 X = -102.6 mm, Y = 123.5 mm, Z = 131.1 mm,       W = 0.0 deg, P = 0.0 deg,
    GP2:
        UF : 1, UT : 2,
       J1 = 0.0 deg, J2 = 0.0 deg
 };
P[160] {
    GP1:
        UF : 6, UT : 5,     CONFIG: 'N U T, 0, 0, 0',
       X = -119.0 mm, Y = 51.8 mm, Z = 131.1 mm,
       W = 0.0 deg, P = 0.0 deg,
    GP2:
        UF : 1, UT : 2,
       J1 = 0.0 deg, J2 = 0.0 deg
 };
P[356] {
    GP1:
        UF : 6, UT : 5,     CONFIG: 'N U T, 0, 0, 0',
 X = -102.0 mm, Y = 122.8 mm, Z = 131.1 mm,       W = 0.0 deg, P = 0.0 deg,
    GP2:
        UF : 1, UT : 2,
       J1 = 0.0 deg, J2 = 0.0 deg
 };
P[161] {
    GP1:
        UF : 6, UT : 5,     CONFIG: 'N U T, 0, 0, 0',
       X = -118.5 mm, Y = 51.0 mm, Z = 131.1 mm,
       W = 0.0 deg, P = 0.0 deg,
    GP2:
        UF : 1, UT : 2,
       J1 = 0.0 deg, J2 = 0.0 deg
 };
P[357] {
    GP1:
        UF : 6, UT : 5,     CONFIG: 'N U T, 0, 0, 0',
 X = -101.5 mm, Y = 122.0 mm, Z = 131.1 mm,       W = 0.0 deg, P = 0.0 deg,
    GP2:
        UF : 1, UT : 2,
       J1 = 0.0 deg, J2 = 0.0 deg
 };
P[162] {
    GP1:
        UF : 6, UT : 5,     CONFIG: 'N U T, 0, 0, 0',
       X = -117.9 mm, Y = 49.9 mm, Z = 131.1 mm,
       W = 0.0 deg, P = 0.0 deg,
    GP2:
        UF : 1, UT : 2,
       J1 = 0.0 deg, J2 = 0.0 deg
 };
P[358] {
    GP1:
        UF : 6, UT : 5,     CONFIG: 'N U T, 0, 0, 0',
 X = -100.9 mm, Y = 120.9 mm, Z = 131.1 mm,       W = 0.0 deg, P = 0.0 deg,
    GP2:
        UF : 1, UT : 2,
       J1 = 0.0 deg, J2 = 0.0 deg
 };
P[163] {
    GP1:
        UF : 6, UT : 5,     CONFIG: 'N U T, 0, 0, 0',
       X = -117.5 mm, Y = 48.5 mm, Z = 131.1 mm,
       W = 0.0 deg, P = 0.0 deg,
    GP2:
        UF : 1, UT : 2,
       J1 = 0.0 deg, J2 = 0.0 deg
 };
P[359] {
    GP1:
        UF : 6, UT : 5,     CONFIG: 'N U T, 0, 0, 0',
 X = -100.5 mm, Y = 119.5 mm, Z = 131.1 mm,       W = 0.0 deg, P = 0.0 deg,
    GP2:
        UF : 1, UT : 2,
       J1 = 0.0 deg, J2 = 0.0 deg
 };
P[164] {
    GP1:
        UF : 6, UT : 5,     CONFIG: 'N U T, 0, 0, 0',
       X = -116.9 mm, Y = 46.0 mm, Z = 131.1 mm,
       W = 0.0 deg, P = 0.0 deg,
    GP2:
        UF : 1, UT : 2,
       J1 = 0.0 deg, J2 = 0.0 deg
 };
P[360] {
    GP1:
        UF : 6, UT : 5,     CONFIG: 'N U T, 0, 0, 0',
 X = -99.9 mm, Y = 117.0 mm, Z = 131.1 mm,       W = 0.0 deg, P = 0.0 deg,
    GP2:
        UF : 1, UT : 2,
       J1 = 0.0 deg, J2 = 0.0 deg
 };
P[165] {
    GP1:
        UF : 6, UT : 5,     CONFIG: 'N U T, 0, 0, 0',
       X = -116.5 mm, Y = 42.8 mm, Z = 131.1 mm,
       W = 0.0 deg, P = 0.0 deg,
    GP2:
        UF : 1, UT : 2,
       J1 = 0.0 deg, J2 = 0.0 deg
 };
P[361] {
    GP1:
        UF : 6, UT : 5,     CONFIG: 'N U T, 0, 0, 0',
 X = -99.5 mm, Y = 113.8 mm, Z = 131.1 mm,       W = 0.0 deg, P = 0.0 deg,
    GP2:
        UF : 1, UT : 2,
       J1 = 0.0 deg, J2 = 0.0 deg
 };
P[166] {
    GP1:
        UF : 6, UT : 5,     CONFIG: 'N U T, 0, 0, 0',
       X = -115.8 mm, Y = 37.9 mm, Z = 131.1 mm,
       W = 0.0 deg, P = 0.0 deg,
    GP2:
        UF : 1, UT : 2,
       J1 = 0.0 deg, J2 = 0.0 deg
 };
P[362] {
    GP1:
        UF : 6, UT : 5,     CONFIG: 'N U T, 0, 0, 0',
 X = -98.8 mm, Y = 108.9 mm, Z = 131.1 mm,       W = 0.0 deg, P = 0.0 deg,
    GP2:
        UF : 1, UT : 2,
       J1 = 0.0 deg, J2 = 0.0 deg
 };
P[167] {
    GP1:
        UF : 6, UT : 5,     CONFIG: 'N U T, 0, 0, 0',
       X = -114.5 mm, Y = 27.9 mm, Z = 131.1 mm,
       W = 0.0 deg, P = 0.0 deg,
    GP2:
        UF : 1, UT : 2,
       J1 = 0.0 deg, J2 = 0.0 deg
 };
P[363] {
    GP1:
        UF : 6, UT : 5,     CONFIG: 'N U T, 0, 0, 0',
 X = -97.5 mm, Y = 98.9 mm, Z = 131.1 mm,       W = 0.0 deg, P = 0.0 deg,
    GP2:
        UF : 1, UT : 2,
       J1 = 0.0 deg, J2 = 0.0 deg
 };
P[168] {
    GP1:
        UF : 6, UT : 5,     CONFIG: 'N U T, 0, 0, 0',
       X = -113.4 mm, Y = 18.0 mm, Z = 131.1 mm,
       W = 0.0 deg, P = 0.0 deg,
    GP2:
        UF : 1, UT : 2,
       J1 = 0.0 deg, J2 = 0.0 deg
 };
P[364] {
    GP1:
        UF : 6, UT : 5,     CONFIG: 'N U T, 0, 0, 0',
 X = -96.4 mm, Y = 89.0 mm, Z = 131.1 mm,       W = 0.0 deg, P = 0.0 deg,
    GP2:
        UF : 1, UT : 2,
       J1 = 0.0 deg, J2 = 0.0 deg
 };
P[169] {
    GP1:
        UF : 6, UT : 5,     CONFIG: 'N U T, 0, 0, 0',
       X = -112.4 mm, Y = 8.1 mm, Z = 131.1 mm,
       W = 0.0 deg, P = 0.0 deg,
    GP2:
        UF : 1, UT : 2,
       J1 = 0.0 deg, J2 = 0.0 deg
 };
P[365] {
    GP1:
        UF : 6, UT : 5,     CONFIG: 'N U T, 0, 0, 0',
 X = -95.4 mm, Y = 79.1 mm, Z = 131.1 mm,       W = 0.0 deg, P = 0.0 deg,
    GP2:
        UF : 1, UT : 2,
       J1 = 0.0 deg, J2 = 0.0 deg
 };
P[170] {
    GP1:
        UF : 6, UT : 5,     CONFIG: 'N U T, 0, 0, 0',
       X = -111.6 mm, Y = -1.9 mm, Z = 131.1 mm,
       W = 0.0 deg, P = 0.0 deg,
    GP2:
        UF : 1, UT : 2,
       J1 = 0.0 deg, J2 = 0.0 deg
 };
P[366] {
    GP1:
        UF : 6, UT : 5,     CONFIG: 'N U T, 0, 0, 0',
 X = -94.6 mm, Y = 69.1 mm, Z = 131.1 mm,       W = 0.0 deg, P = 0.0 deg,
    GP2:
        UF : 1, UT : 2,
       J1 = 0.0 deg, J2 = 0.0 deg
 };
P[171] {
    GP1:
        UF : 6, UT : 5,     CONFIG: 'N U T, 0, 0, 0',
       X = -110.9 mm, Y = -11.9 mm, Z = 131.1 mm,
       W = 0.0 deg, P = 0.0 deg,
    GP2:
        UF : 1, UT : 2,
       J1 = 0.0 deg, J2 = 0.0 deg
 };
P[367] {
    GP1:
        UF : 6, UT : 5,     CONFIG: 'N U T, 0, 0, 0',
 X = -93.9 mm, Y = 59.1 mm, Z = 131.1 mm,       W = 0.0 deg, P = 0.0 deg,
    GP2:
        UF : 1, UT : 2,
       J1 = 0.0 deg, J2 = 0.0 deg
 };
P[172] {
    GP1:
        UF : 6, UT : 5,     CONFIG: 'N U T, 0, 0, 0',
       X = -110.3 mm, Y = -21.9 mm, Z = 131.1 mm,
       W = 0.0 deg, P = 0.0 deg,
    GP2:
        UF : 1, UT : 2,
       J1 = 0.0 deg, J2 = 0.0 deg
 };
P[368] {
    GP1:
        UF : 6, UT : 5,     CONFIG: 'N U T, 0, 0, 0',
 X = -93.3 mm, Y = 49.1 mm, Z = 131.1 mm,       W = 0.0 deg, P = 0.0 deg,
    GP2:
        UF : 1, UT : 2,
       J1 = 0.0 deg, J2 = 0.0 deg
 };
P[173] {
    GP1:
        UF : 6, UT : 5,     CONFIG: 'N U T, 0, 0, 0',
       X = -110.1 mm, Y = -24.0 mm, Z = 131.1 mm,
       W = 0.0 deg, P = 0.0 deg,
    GP2:
        UF : 1, UT : 2,
       J1 = 0.0 deg, J2 = 0.0 deg
 };
P[369] {
    GP1:
        UF : 6, UT : 5,     CONFIG: 'N U T, 0, 0, 0',
 X = -93.1 mm, Y = 47.0 mm, Z = 131.1 mm,       W = 0.0 deg, P = 0.0 deg,
    GP2:
        UF : 1, UT : 2,
       J1 = 0.0 deg, J2 = 0.0 deg
 };
P[174] {
    GP1:
        UF : 6, UT : 5,     CONFIG: 'N U T, 0, 0, 0',
       X = -109.5 mm, Y = -26.0 mm, Z = 131.1 mm,
       W = 0.0 deg, P = 0.0 deg,
    GP2:
        UF : 1, UT : 2,
       J1 = 0.0 deg, J2 = 0.0 deg
 };
P[370] {
    GP1:
        UF : 6, UT : 5,     CONFIG: 'N U T, 0, 0, 0',
 X = -92.5 mm, Y = 45.0 mm, Z = 131.1 mm,       W = 0.0 deg, P = 0.0 deg,
    GP2:
        UF : 1, UT : 2,
       J1 = 0.0 deg, J2 = 0.0 deg
 };
P[175] {
    GP1:
        UF : 6, UT : 5,     CONFIG: 'N U T, 0, 0, 0',
       X = -108.7 mm, Y = -28.0 mm, Z = 131.1 mm,
       W = 0.0 deg, P = 0.0 deg,
    GP2:
        UF : 1, UT : 2,
       J1 = 0.0 deg, J2 = 0.0 deg
 };
P[371] {
    GP1:
        UF : 6, UT : 5,     CONFIG: 'N U T, 0, 0, 0',
 X = -91.7 mm, Y = 43.0 mm, Z = 131.1 mm,       W = 0.0 deg, P = 0.0 deg,
    GP2:
        UF : 1, UT : 2,
       J1 = 0.0 deg, J2 = 0.0 deg
 };
P[176] {
    GP1:
        UF : 6, UT : 5,     CONFIG: 'N U T, 0, 0, 0',
       X = -107.0 mm, Y = -30.9 mm, Z = 131.1 mm,
       W = 0.0 deg, P = 0.0 deg,
    GP2:
        UF : 1, UT : 2,
       J1 = 0.0 deg, J2 = 0.0 deg
 };
P[372] {
    GP1:
        UF : 6, UT : 5,     CONFIG: 'N U T, 0, 0, 0',
 X = -90.0 mm, Y = 40.1 mm, Z = 131.1 mm,       W = 0.0 deg, P = 0.0 deg,
    GP2:
        UF : 1, UT : 2,
       J1 = 0.0 deg, J2 = 0.0 deg
 };
P[177] {
    GP1:
        UF : 6, UT : 5,     CONFIG: 'N U T, 0, 0, 0',
       X = -103.8 mm, Y = -36.3 mm, Z = 131.1 mm,
       W = 0.0 deg, P = 0.0 deg,
    GP2:
        UF : 1, UT : 2,
       J1 = 0.0 deg, J2 = 0.0 deg
 };
P[373] {
    GP1:
        UF : 6, UT : 5,     CONFIG: 'N U T, 0, 0, 0',
 X = -86.8 mm, Y = 34.7 mm, Z = 131.1 mm,       W = 0.0 deg, P = 0.0 deg,
    GP2:
        UF : 1, UT : 2,
       J1 = 0.0 deg, J2 = 0.0 deg
 };
P[178] {
    GP1:
        UF : 6, UT : 5,     CONFIG: 'N U T, 0, 0, 0',
       X = -102.7 mm, Y = -38.0 mm, Z = 131.1 mm,
       W = 0.0 deg, P = 0.0 deg,
    GP2:
        UF : 1, UT : 2,
       J1 = 0.0 deg, J2 = 0.0 deg
 };
P[374] {
    GP1:
        UF : 6, UT : 5,     CONFIG: 'N U T, 0, 0, 0',
 X = -85.7 mm, Y = 33.0 mm, Z = 131.1 mm,       W = 0.0 deg, P = 0.0 deg,
    GP2:
        UF : 1, UT : 2,
       J1 = 0.0 deg, J2 = 0.0 deg
 };
P[179] {
    GP1:
        UF : 6, UT : 5,     CONFIG: 'N U T, 0, 0, 0',
       X = -101.2 mm, Y = -39.4 mm, Z = 131.1 mm,
       W = 0.0 deg, P = 0.0 deg,
    GP2:
        UF : 1, UT : 2,
       J1 = 0.0 deg, J2 = 0.0 deg
 };
P[375] {
    GP1:
        UF : 6, UT : 5,     CONFIG: 'N U T, 0, 0, 0',
 X = -84.2 mm, Y = 31.6 mm, Z = 131.1 mm,       W = 0.0 deg, P = 0.0 deg,
    GP2:
        UF : 1, UT : 2,
       J1 = 0.0 deg, J2 = 0.0 deg
 };
P[180] {
    GP1:
        UF : 6, UT : 5,     CONFIG: 'N U T, 0, 0, 0',
       X = -99.8 mm, Y = -40.1 mm, Z = 131.1 mm,
       W = 0.0 deg, P = 0.0 deg,
    GP2:
        UF : 1, UT : 2,
       J1 = 0.0 deg, J2 = 0.0 deg
 };
P[376] {
    GP1:
        UF : 6, UT : 5,     CONFIG: 'N U T, 0, 0, 0',
 X = -82.8 mm, Y = 30.9 mm, Z = 131.1 mm,       W = 0.0 deg, P = 0.0 deg,
    GP2:
        UF : 1, UT : 2,
       J1 = 0.0 deg, J2 = 0.0 deg
 };
P[181] {
    GP1:
        UF : 6, UT : 5,     CONFIG: 'N U T, 0, 0, 0',
       X = -98.3 mm, Y = -40.7 mm, Z = 131.1 mm,
       W = 0.0 deg, P = 0.0 deg,
    GP2:
        UF : 1, UT : 2,
       J1 = 0.0 deg, J2 = 0.0 deg
 };
P[377] {
    GP1:
        UF : 6, UT : 5,     CONFIG: 'N U T, 0, 0, 0',
 X = -81.3 mm, Y = 30.3 mm, Z = 131.1 mm,       W = 0.0 deg, P = 0.0 deg,
    GP2:
        UF : 1, UT : 2,
       J1 = 0.0 deg, J2 = 0.0 deg
 };
P[182] {
    GP1:
        UF : 6, UT : 5,     CONFIG: 'N U T, 0, 0, 0',
       X = -96.7 mm, Y = -40.8 mm, Z = 131.1 mm,
       W = 0.0 deg, P = 0.0 deg,
    GP2:
        UF : 1, UT : 2,
       J1 = 0.0 deg, J2 = 0.0 deg
 };
P[378] {
    GP1:
        UF : 6, UT : 5,     CONFIG: 'N U T, 0, 0, 0',
 X = -79.7 mm, Y = 30.2 mm, Z = 131.1 mm,       W = 0.0 deg, P = 0.0 deg,
    GP2:
        UF : 1, UT : 2,
       J1 = 0.0 deg, J2 = 0.0 deg
 };
P[183] {
    GP1:
        UF : 6, UT : 5,     CONFIG: 'N U T, 0, 0, 0',
       X = -95.2 mm, Y = -40.7 mm, Z = 131.1 mm,
       W = 0.0 deg, P = 0.0 deg,
    GP2:
        UF : 1, UT : 2,
       J1 = 0.0 deg, J2 = 0.0 deg
 };
P[379] {
    GP1:
        UF : 6, UT : 5,     CONFIG: 'N U T, 0, 0, 0',
 X = -78.2 mm, Y = 30.3 mm, Z = 131.1 mm,       W = 0.0 deg, P = 0.0 deg,
    GP2:
        UF : 1, UT : 2,
       J1 = 0.0 deg, J2 = 0.0 deg
 };
P[184] {
    GP1:
        UF : 6, UT : 5,     CONFIG: 'N U T, 0, 0, 0',
       X = -93.7 mm, Y = -40.3 mm, Z = 131.1 mm,
       W = 0.0 deg, P = 0.0 deg,
    GP2:
        UF : 1, UT : 2,
       J1 = 0.0 deg, J2 = 0.0 deg
 };
P[380] {
    GP1:
        UF : 6, UT : 5,     CONFIG: 'N U T, 0, 0, 0',
 X = -76.7 mm, Y = 30.7 mm, Z = 131.1 mm,       W = 0.0 deg, P = 0.0 deg,
    GP2:
        UF : 1, UT : 2,
       J1 = 0.0 deg, J2 = 0.0 deg
 };
P[185] {
    GP1:
        UF : 6, UT : 5,     CONFIG: 'N U T, 0, 0, 0',
       X = -92.2 mm, Y = -39.6 mm, Z = 131.1 mm,
       W = 0.0 deg, P = 0.0 deg,
    GP2:
        UF : 1, UT : 2,
       J1 = 0.0 deg, J2 = 0.0 deg
 };
P[381] {
    GP1:
        UF : 6, UT : 5,     CONFIG: 'N U T, 0, 0, 0',
 X = -75.2 mm, Y = 31.4 mm, Z = 131.1 mm,       W = 0.0 deg, P = 0.0 deg,
    GP2:
        UF : 1, UT : 2,
       J1 = 0.0 deg, J2 = 0.0 deg
 };
P[186] {
    GP1:
        UF : 6, UT : 5,     CONFIG: 'N U T, 0, 0, 0',
       X = -87.3 mm, Y = -36.9 mm, Z = 131.1 mm,
       W = 0.0 deg, P = 0.0 deg,
    GP2:
        UF : 1, UT : 2,
       J1 = 0.0 deg, J2 = 0.0 deg
 };
P[382] {
    GP1:
        UF : 6, UT : 5,     CONFIG: 'N U T, 0, 0, 0',
 X = -70.3 mm, Y = 34.1 mm, Z = 131.1 mm,       W = 0.0 deg, P = 0.0 deg,
    GP2:
        UF : 1, UT : 2,
       J1 = 0.0 deg, J2 = 0.0 deg
 };
P[187] {
    GP1:
        UF : 6, UT : 5,     CONFIG: 'N U T, 0, 0, 0',
       X = -78.5 mm, Y = -32.1 mm, Z = 131.1 mm,
       W = 0.0 deg, P = 0.0 deg,
    GP2:
        UF : 1, UT : 2,
       J1 = 0.0 deg, J2 = 0.0 deg
 };
P[383] {
    GP1:
        UF : 6, UT : 5,     CONFIG: 'N U T, 0, 0, 0',
 X = -61.5 mm, Y = 38.9 mm, Z = 131.1 mm,       W = 0.0 deg, P = 0.0 deg,
    GP2:
        UF : 1, UT : 2,
       J1 = 0.0 deg, J2 = 0.0 deg
 };
P[188] {
    GP1:
        UF : 6, UT : 5,     CONFIG: 'N U T, 0, 0, 0',
       X = -69.8 mm, Y = -27.2 mm, Z = 131.1 mm,
       W = 0.0 deg, P = 0.0 deg,
    GP2:
        UF : 1, UT : 2,
       J1 = 0.0 deg, J2 = 0.0 deg
 };
P[384] {
    GP1:
        UF : 6, UT : 5,     CONFIG: 'N U T, 0, 0, 0',
 X = -52.8 mm, Y = 43.8 mm, Z = 131.1 mm,       W = 0.0 deg, P = 0.0 deg,
    GP2:
        UF : 1, UT : 2,
       J1 = 0.0 deg, J2 = 0.0 deg
 };
P[189] {
    GP1:
        UF : 6, UT : 5,     CONFIG: 'N U T, 0, 0, 0',
       X = -61.0 mm, Y = -22.4 mm, Z = 131.1 mm,
       W = 0.0 deg, P = 0.0 deg,
    GP2:
        UF : 1, UT : 2,
       J1 = 0.0 deg, J2 = 0.0 deg
 };
P[385] {
    GP1:
        UF : 6, UT : 5,     CONFIG: 'N U T, 0, 0, 0',
 X = -44.0 mm, Y = 48.6 mm, Z = 131.1 mm,       W = 0.0 deg, P = 0.0 deg,
    GP2:
        UF : 1, UT : 2,
       J1 = 0.0 deg, J2 = 0.0 deg
 };
P[190] {
    GP1:
        UF : 6, UT : 5,     CONFIG: 'N U T, 0, 0, 0',
       X = -52.3 mm, Y = -17.6 mm, Z = 131.1 mm,
       W = 0.0 deg, P = 0.0 deg,
    GP2:
        UF : 1, UT : 2,
       J1 = 0.0 deg, J2 = 0.0 deg
 };
P[386] {
    GP1:
        UF : 6, UT : 5,     CONFIG: 'N U T, 0, 0, 0',
 X = -35.3 mm, Y = 53.4 mm, Z = 131.1 mm,       W = 0.0 deg, P = 0.0 deg,
    GP2:
        UF : 1, UT : 2,
       J1 = 0.0 deg, J2 = 0.0 deg
 };
P[191] {
    GP1:
        UF : 6, UT : 5,     CONFIG: 'N U T, 0, 0, 0',
       X = -43.6 mm, Y = -12.7 mm, Z = 131.1 mm,
       W = 0.0 deg, P = 0.0 deg,
    GP2:
        UF : 1, UT : 2,
       J1 = 0.0 deg, J2 = 0.0 deg
 };
P[387] {
    GP1:
        UF : 6, UT : 5,     CONFIG: 'N U T, 0, 0, 0',
 X = -26.6 mm, Y = 58.3 mm, Z = 131.1 mm,       W = 0.0 deg, P = 0.0 deg,
    GP2:
        UF : 1, UT : 2,
       J1 = 0.0 deg, J2 = 0.0 deg
 };
P[192] {
    GP1:
        UF : 6, UT : 5,     CONFIG: 'N U T, 0, 0, 0',
       X = -34.8 mm, Y = -7.9 mm, Z = 131.1 mm,
       W = 0.0 deg, P = 0.0 deg,
    GP2:
        UF : 1, UT : 2,
       J1 = 0.0 deg, J2 = 0.0 deg
 };
P[388] {
    GP1:
        UF : 6, UT : 5,     CONFIG: 'N U T, 0, 0, 0',
 X = -17.8 mm, Y = 63.1 mm, Z = 131.1 mm,       W = 0.0 deg, P = 0.0 deg,
    GP2:
        UF : 1, UT : 2,
       J1 = 0.0 deg, J2 = 0.0 deg
 };
P[193] {
    GP1:
        UF : 6, UT : 5,     CONFIG: 'N U T, 0, 0, 0',
       X = -26.1 mm, Y = -3.0 mm, Z = 131.1 mm,
       W = 0.0 deg, P = 0.0 deg,
    GP2:
        UF : 1, UT : 2,
       J1 = 0.0 deg, J2 = 0.0 deg
 };
P[389] {
    GP1:
        UF : 6, UT : 5,     CONFIG: 'N U T, 0, 0, 0',
 X = -9.1 mm, Y = 68.0 mm, Z = 131.1 mm,       W = 0.0 deg, P = 0.0 deg,
    GP2:
        UF : 1, UT : 2,
       J1 = 0.0 deg, J2 = 0.0 deg
 };
P[194] {
    GP1:
        UF : 6, UT : 5,     CONFIG: 'N U T, 0, 0, 0',
       X = -17.3 mm, Y = 1.8 mm, Z = 131.1 mm,
       W = 0.0 deg, P = 0.0 deg,
    GP2:
        UF : 1, UT : 2,
       J1 = 0.0 deg, J2 = 0.0 deg
 };
P[390] {
    GP1:
        UF : 6, UT : 5,     CONFIG: 'N U T, 0, 0, 0',
 X = -0.3 mm, Y = 72.8 mm, Z = 131.1 mm,       W = 0.0 deg, P = 0.0 deg,
    GP2:
        UF : 1, UT : 2,
       J1 = 0.0 deg, J2 = 0.0 deg
 };
/END
